// Mitsubishi GX Works2 project: Tetris_20220329   PLC: Q03UDV

PROGRAM 94_TOOLS  // Common Tools
; [Title]P1030 Calculate 16's Field Address
      P1030
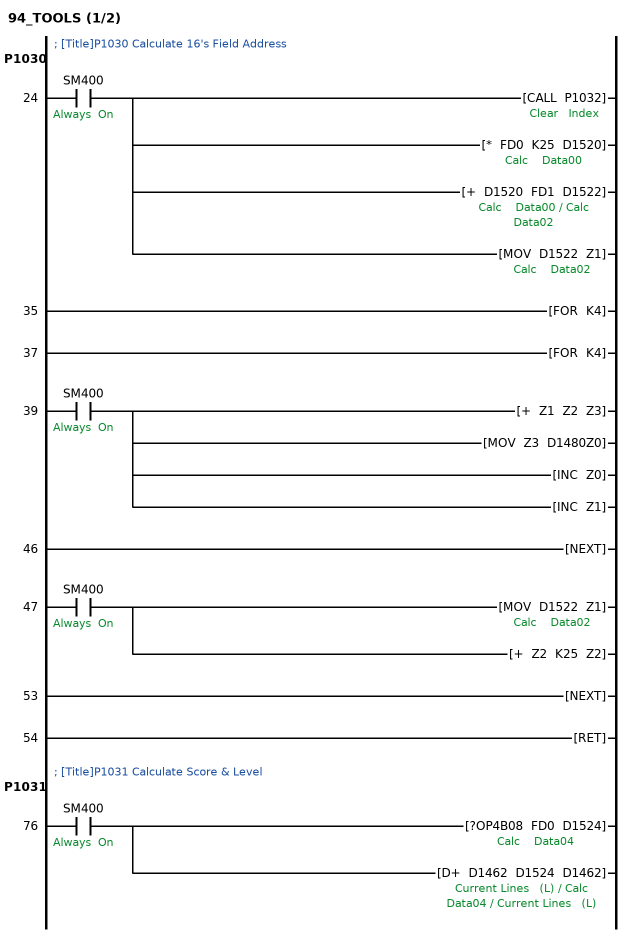
24    LD      SM400  ; Always  On
      CALL    P1032  ; Clear   Index
      *       FD0 K25 D1520  ; Calc    Data00
      +       D1520 FD1 D1522  ; Calc    Data02
      MOV     D1522 Z1
35    FOR     K4
37    FOR     K4
39    LD      SM400  ; Always  On
      +       Z1 Z2 Z3
      MOV     Z3 D1480Z0
      INC     Z0
      INC     Z1
46    NEXT
47    LD      SM400  ; Always  On
      MOV     D1522 Z1
      +       Z2 K25 Z2
53    NEXT
54    RET
; [Title]P1031 Calculate Score & Level
      P1031
76    LD      SM400  ; Always  On
      ?OP4B08 FD0 D1524  ; Calc    Data04
      D+      D1462 D1524 D1462  ; Current Lines   (L)
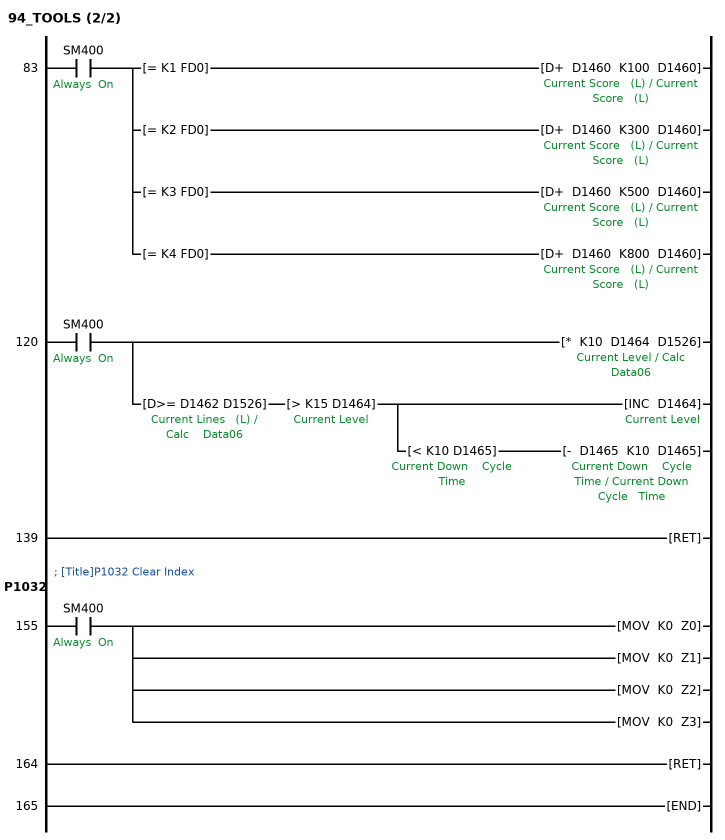
83    LD      SM400  ; Always  On
      MPS
      AND=    K1 FD0
      D+      D1460 K100 D1460  ; Current Score   (L)
      MRD
      AND=    K2 FD0
      D+      D1460 K300 D1460
      MRD
      AND=    K3 FD0
      D+      D1460 K500 D1460
      MPP
      AND=    K4 FD0
      D+      D1460 K800 D1460
120   LD      SM400  ; Always  On
      *       K10 D1464 D1526  ; Current Level / Calc    Data06
      ANDD>=  D1462 D1526  ; Current Lines   (L) / Calc    Data06
      AND>    K15 D1464  ; Current Level
      INC     D1464
      AND<    K10 D1465  ; Current Down    Cycle   Time
      -       D1465 K10 D1465
139   RET
; [Title]P1032 Clear Index
      P1032
155   LD      SM400  ; Always  On
      MOV     K0 Z0
      MOV     K0 Z1
      MOV     K0 Z2
      MOV     K0 Z3
164   RET
165   END
END_PROGRAM

PROGRAM 02_GAME  // Main Game Control
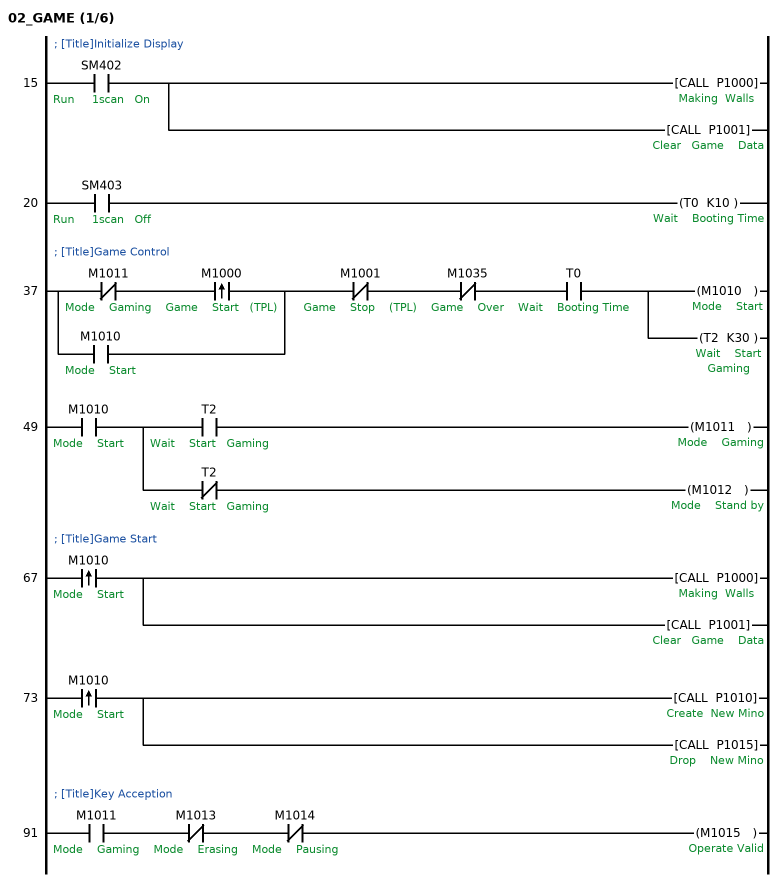
; [Title]Initialize Display
15    LD      SM402  ; Run     1scan   On
      CALL    P1000  ; Making  Walls
      CALL    P1001  ; Clear   Game    Data
20    LD      SM403  ; Run     1scan   Off
      OUT     T0 K10  ; Wait    Booting Time
; [Title]Game Control
37    LDI     M1011  ; Mode    Gaming
      ANDP    M1000  ; Game    Start   (TPL)
      OR      M1010  ; Mode    Start
      ANI     M1001  ; Game    Stop    (TPL)
      ANI     M1035  ; Game    Over
      AND     T0  ; Wait    Booting Time
      OUT     M1010  ; Mode    Start
      OUT     T2 K30  ; Wait    Start   Gaming
49    LD      M1010  ; Mode    Start
      MPS
      AND     T2  ; Wait    Start   Gaming
      OUT     M1011  ; Mode    Gaming
      MPP
      ANI     T2  ; Wait    Start   Gaming
      OUT     M1012  ; Mode    Stand by
; [Title]Game Start
67    LDP     M1010  ; Mode    Start
      CALL    P1000
      CALL    P1001
73    LDP     M1010  ; Mode    Start
      CALL    P1010  ; Create  New Mino
      CALL    P1015  ; Drop    New Mino
; [Title]Key Acception
91    LD      M1011  ; Mode    Gaming
      ANI     M1013  ; Mode    Erasing
      ANI     M1014  ; Mode    Pausing
      OUT     M1015  ; Operate Valid
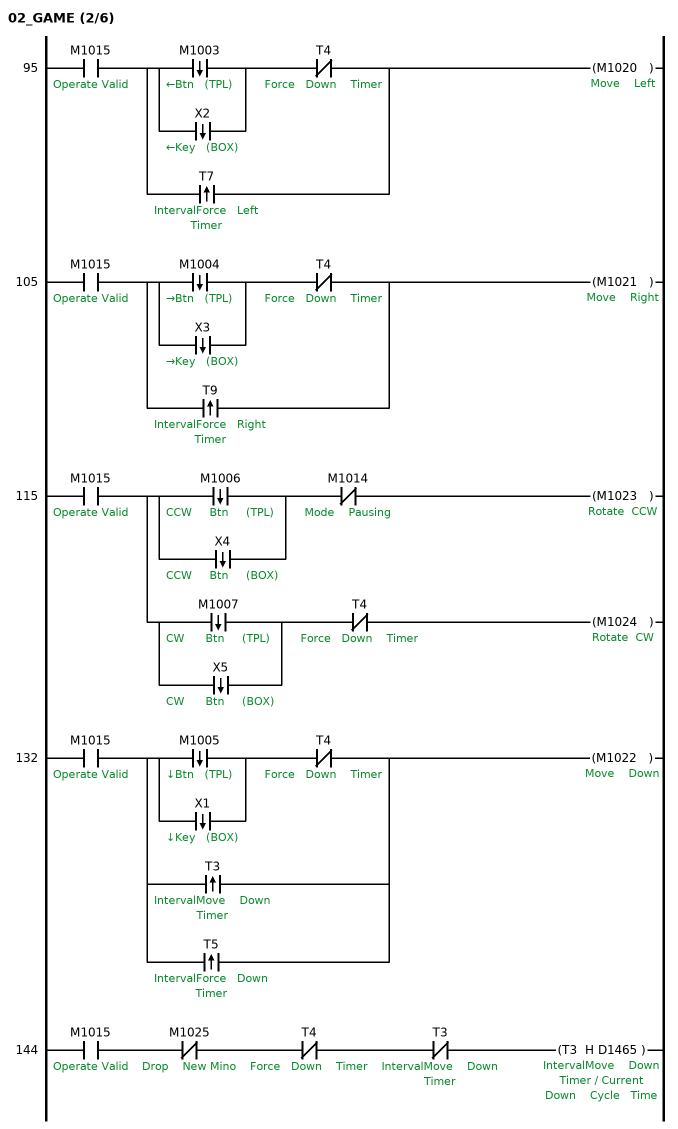
95    LD      M1015  ; Operate Valid
      LDF     M1003  ; ←Btn   (TPL)
      ORF     X2  ; ←Key   (BOX)
      ANI     T4  ; Force   Down    Timer
      ORP     T7  ; IntervalForce   Left    Timer
      ANB
      OUT     M1020  ; Move    Left
105   LD      M1015  ; Operate Valid
      LDF     M1004  ; →Btn   (TPL)
      ORF     X3  ; →Key   (BOX)
      ANI     T4  ; Force   Down    Timer
      ORP     T9  ; IntervalForce   Right   Timer
      ANB
      OUT     M1021  ; Move    Right
115   LD      M1015  ; Operate Valid
      MPS
      LDF     M1006  ; CCW     Btn     (TPL)
      ORF     X4  ; CCW     Btn     (BOX)
      ANB
      ANI     M1014  ; Mode    Pausing
      OUT     M1023  ; Rotate  CCW
      MPP
      LDF     M1007  ; CW      Btn     (TPL)
      ORF     X5  ; CW      Btn     (BOX)
      ANB
      ANI     T4  ; Force   Down    Timer
      OUT     M1024  ; Rotate  CW
132   LD      M1015  ; Operate Valid
      LDF     M1005  ; ↓Btn   (TPL)
      ORF     X1  ; ↓Key   (BOX)
      ANI     T4  ; Force   Down    Timer
      ORP     T3  ; IntervalMove    Down    Timer
      ORP     T5  ; IntervalForce   Down    Timer
      ANB
      OUT     M1022  ; Move    Down
144   LD      M1015  ; Operate Valid
      ANI     M1025  ; Drop    New Mino
      ANI     T4  ; Force   Down    Timer
      ANI     T3  ; IntervalMove    Down    Timer
      OUTH    T3 D1465  ; IntervalMove    Down    Timer / Current Down    Cycle   Time
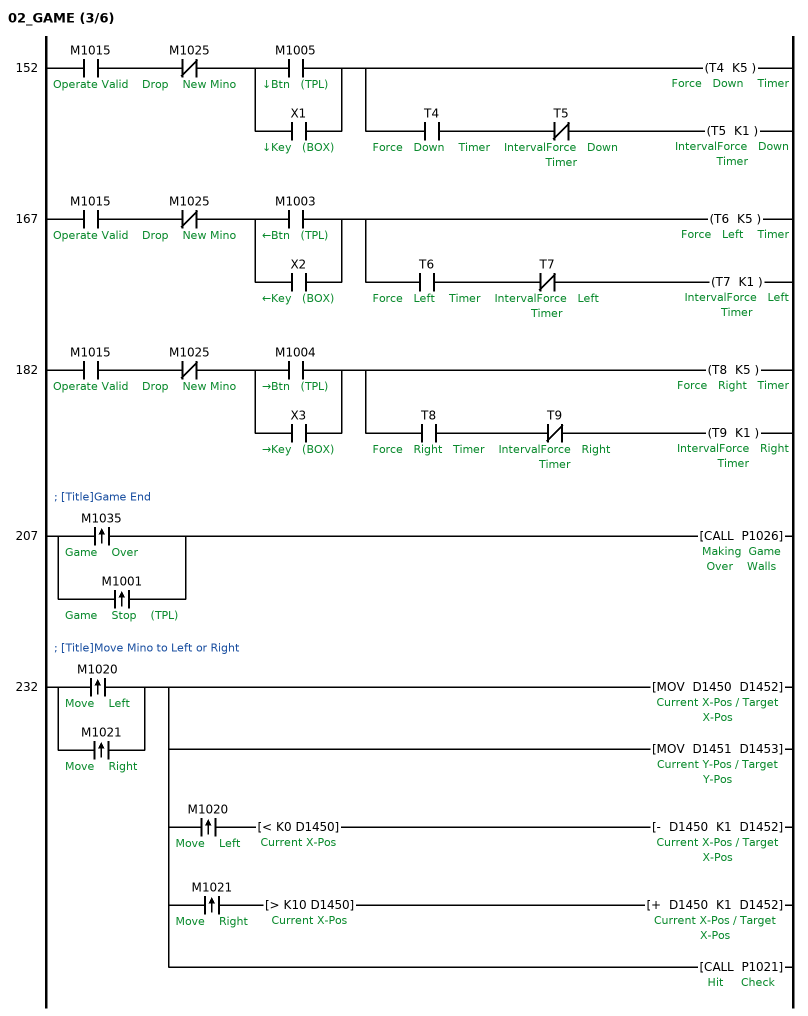
152   LD      M1015  ; Operate Valid
      ANI     M1025  ; Drop    New Mino
      LD      M1005  ; ↓Btn   (TPL)
      OR      X1  ; ↓Key   (BOX)
      ANB
      OUT     T4 K5  ; Force   Down    Timer
      AND     T4  ; Force   Down    Timer
      ANI     T5  ; IntervalForce   Down    Timer
      OUT     T5 K1  ; IntervalForce   Down    Timer
167   LD      M1015  ; Operate Valid
      ANI     M1025  ; Drop    New Mino
      LD      M1003  ; ←Btn   (TPL)
      OR      X2  ; ←Key   (BOX)
      ANB
      OUT     T6 K5  ; Force   Left    Timer
      AND     T6  ; Force   Left    Timer
      ANI     T7  ; IntervalForce   Left    Timer
      OUT     T7 K1  ; IntervalForce   Left    Timer
182   LD      M1015  ; Operate Valid
      ANI     M1025  ; Drop    New Mino
      LD      M1004  ; →Btn   (TPL)
      OR      X3  ; →Key   (BOX)
      ANB
      OUT     T8 K5  ; Force   Right   Timer
      AND     T8  ; Force   Right   Timer
      ANI     T9  ; IntervalForce   Right   Timer
      OUT     T9 K1  ; IntervalForce   Right   Timer
; [Title]Game End
207   LDP     M1035  ; Game    Over
      ORP     M1001  ; Game    Stop    (TPL)
      CALL    P1026  ; Making  Game    Over    Walls
; [Title]Move Mino to Left or Right
232   LDP     M1020  ; Move    Left
      ORP     M1021  ; Move    Right
      MOV     D1450 D1452  ; Current X-Pos / Target  X-Pos
      MOV     D1451 D1453  ; Current Y-Pos / Target  Y-Pos
      MPS
      ANDP    M1020  ; Move    Left
      AND<    K0 D1450  ; Current X-Pos
      -       D1450 K1 D1452
      MRD
      ANDP    M1021  ; Move    Right
      AND>    K10 D1450  ; Current X-Pos
      +       D1450 K1 D1452
      MPP
      CALL    P1021  ; Hit     Check
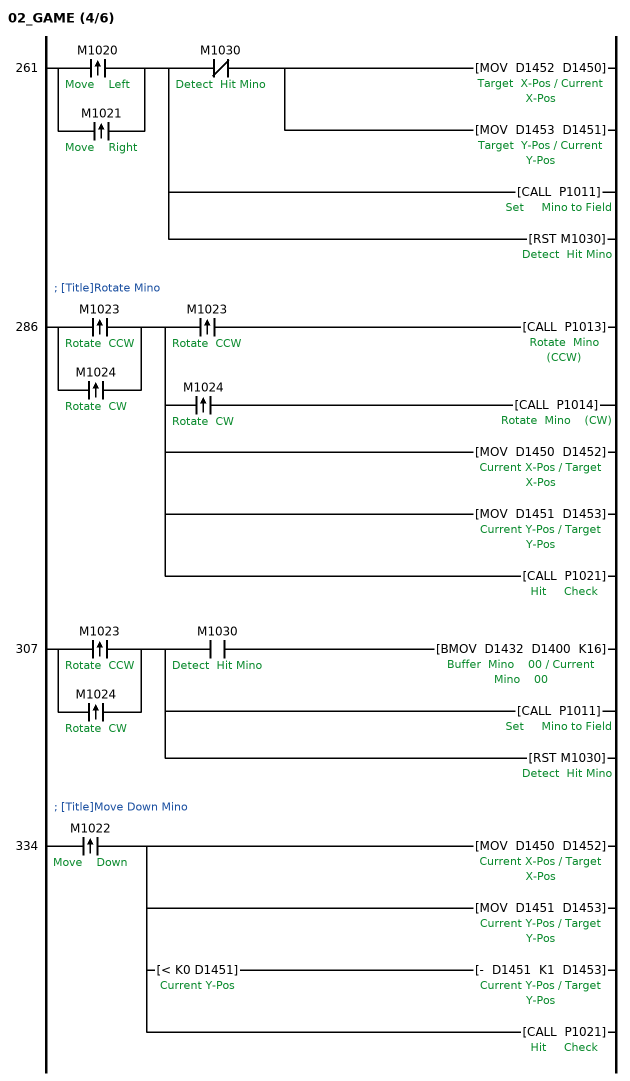
261   LDP     M1020  ; Move    Left
      ORP     M1021  ; Move    Right
      MPS
      ANI     M1030  ; Detect  Hit Mino
      MOV     D1452 D1450
      MOV     D1453 D1451
      MPP
      CALL    P1011  ; Set     Mino to Field
      RST     M1030  ; Detect  Hit Mino
; [Title]Rotate Mino
286   LDP     M1023  ; Rotate  CCW
      ORP     M1024  ; Rotate  CW
      MPS
      ANDP    M1023  ; Rotate  CCW
      CALL    P1013  ; Rotate  Mino    (CCW)
      MRD
      ANDP    M1024  ; Rotate  CW
      CALL    P1014  ; Rotate  Mino    (CW)
      MPP
      MOV     D1450 D1452
      MOV     D1451 D1453
      CALL    P1021
307   LDP     M1023  ; Rotate  CCW
      ORP     M1024  ; Rotate  CW
      MPS
      AND     M1030  ; Detect  Hit Mino
      BMOV    D1432 D1400 K16  ; Buffer  Mino    00 / Current Mino    00
      MPP
      CALL    P1011
      RST     M1030  ; Detect  Hit Mino
; [Title]Move Down Mino
334   LDP     M1022  ; Move    Down
      MOV     D1450 D1452
      MOV     D1451 D1453
      MPS
      AND<    K0 D1451  ; Current Y-Pos
      -       D1451 K1 D1453
      MPP
      CALL    P1021
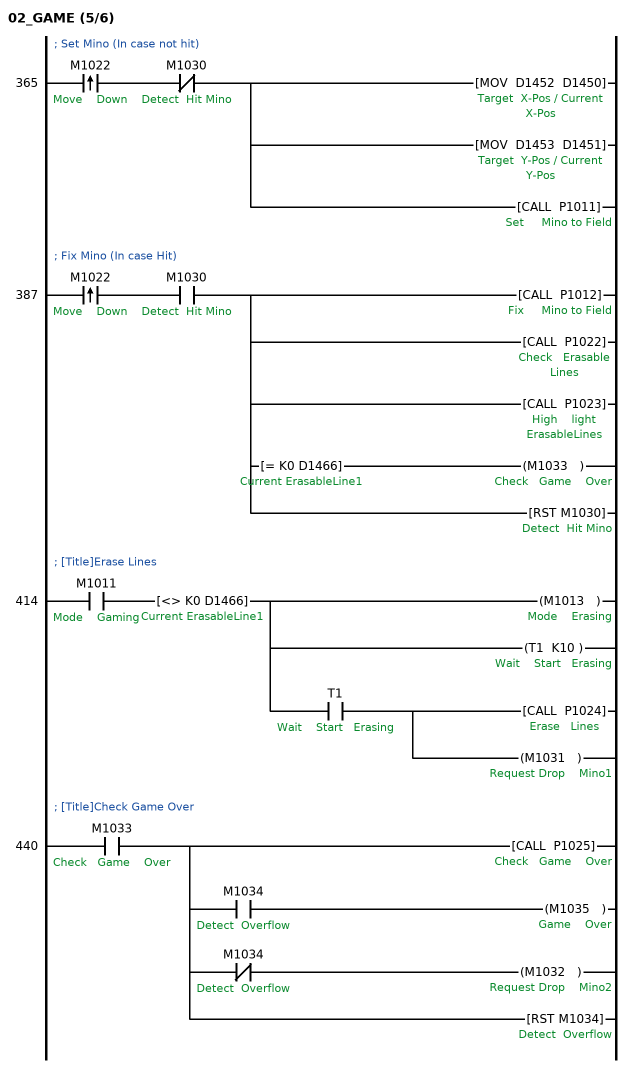
; Set Mino (In case not hit)
365   LDP     M1022  ; Move    Down
      ANI     M1030  ; Detect  Hit Mino
      MOV     D1452 D1450
      MOV     D1453 D1451
      CALL    P1011
; Fix Mino (In case Hit)
387   LDP     M1022  ; Move    Down
      AND     M1030  ; Detect  Hit Mino
      CALL    P1012  ; Fix     Mino to Field
      CALL    P1022  ; Check   ErasableLines
      CALL    P1023  ; High    light   ErasableLines
      MPS
      AND=    K0 D1466  ; Current ErasableLine1
      OUT     M1033  ; Check   Game    Over
      MPP
      RST     M1030  ; Detect  Hit Mino
; [Title]Erase Lines
414   LD      M1011  ; Mode    Gaming
      AND<>   K0 D1466  ; Current ErasableLine1
      OUT     M1013  ; Mode    Erasing
      OUT     T1 K10  ; Wait    Start   Erasing
      AND     T1  ; Wait    Start   Erasing
      CALL    P1024  ; Erase   Lines
      OUT     M1031  ; Request Drop    Mino1
; [Title]Check Game Over
440   LD      M1033  ; Check   Game    Over
      CALL    P1025  ; Check   Game    Over
      MPS
      AND     M1034  ; Detect  Overflow
      OUT     M1035  ; Game    Over
      MRD
      ANI     M1034  ; Detect  Overflow
      OUT     M1032  ; Request Drop    Mino2
      MPP
      RST     M1034  ; Detect  Overflow
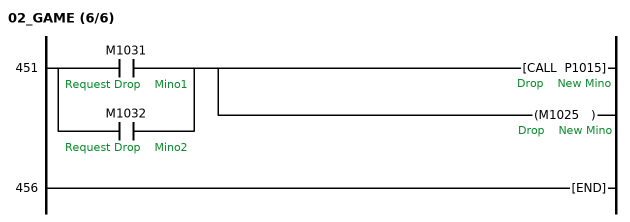
451   LD      M1031  ; Request Drop    Mino1
      OR      M1032  ; Request Drop    Mino2
      CALL    P1015
      OUT     M1025  ; Drop    New Mino
456   END
END_PROGRAM

PROGRAM 91_SETUP  // Setup Condition
; [Title]P1000 Making Walls
; Make Walls and Clear Field
      P1000
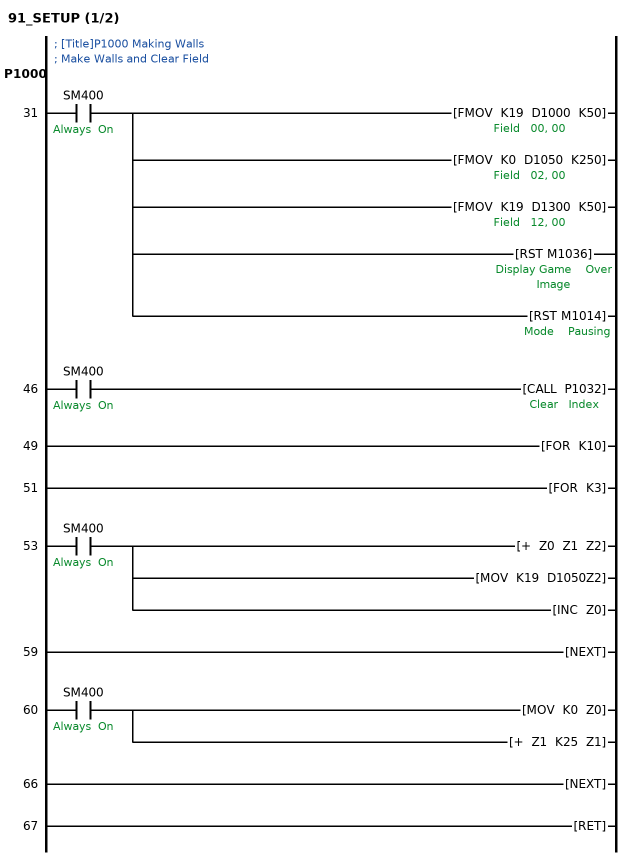
31    LD      SM400  ; Always  On
      FMOV    K19 D1000 K50  ; Field   00, 00
      FMOV    K0 D1050 K250  ; Field   02, 00
      FMOV    K19 D1300 K50  ; Field   12, 00
      RST     M1036  ; Display Game    Over    Image
      RST     M1014  ; Mode    Pausing
46    LD      SM400  ; Always  On
      CALL    P1032  ; Clear   Index
49    FOR     K10
51    FOR     K3
53    LD      SM400  ; Always  On
      +       Z0 Z1 Z2
      MOV     K19 D1050Z2
      INC     Z0
59    NEXT
60    LD      SM400  ; Always  On
      MOV     K0 Z0
      +       Z1 K25 Z1
66    NEXT
67    RET
; [Title]P1001 Clear All Game Data
      P1001
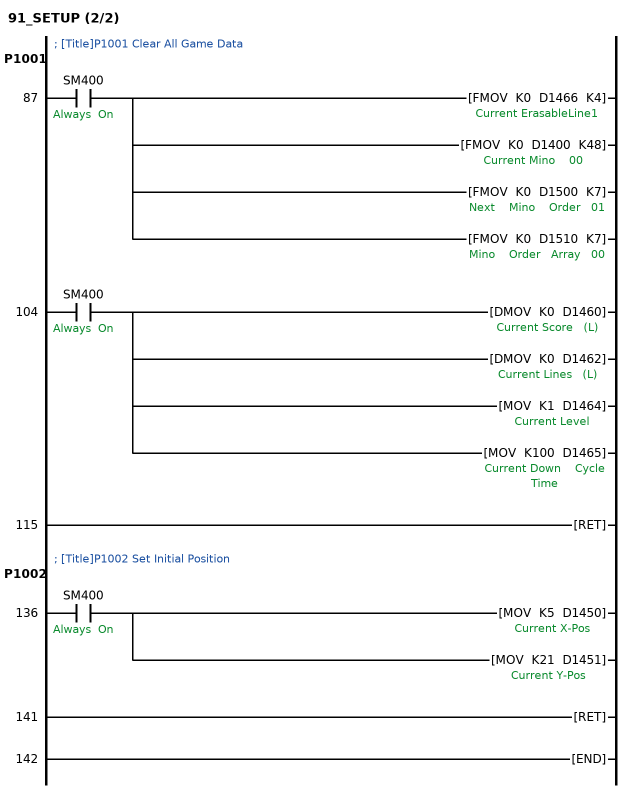
87    LD      SM400  ; Always  On
      FMOV    K0 D1466 K4  ; Current ErasableLine1
      FMOV    K0 D1400 K48  ; Current Mino    00
      FMOV    K0 D1500 K7  ; Next    Mino    Order   01
      FMOV    K0 D1510 K7  ; Mino    Order   Array   00
104   LD      SM400  ; Always  On
      DMOV    K0 D1460  ; Current Score   (L)
      DMOV    K0 D1462  ; Current Lines   (L)
      MOV     K1 D1464  ; Current Level
      MOV     K100 D1465  ; Current Down    Cycle   Time
115   RET
; [Title]P1002 Set Initial Position
      P1002
136   LD      SM400  ; Always  On
      MOV     K5 D1450  ; Current X-Pos
      MOV     K21 D1451  ; Current Y-Pos
141   RET
142   END
END_PROGRAM

PROGRAM 92_MINO  // Manage Mino
; [Title]P1010 Create New Mino
; Make New Mino Order & Copy Mino Data to Reserve Mino Area
      P1010
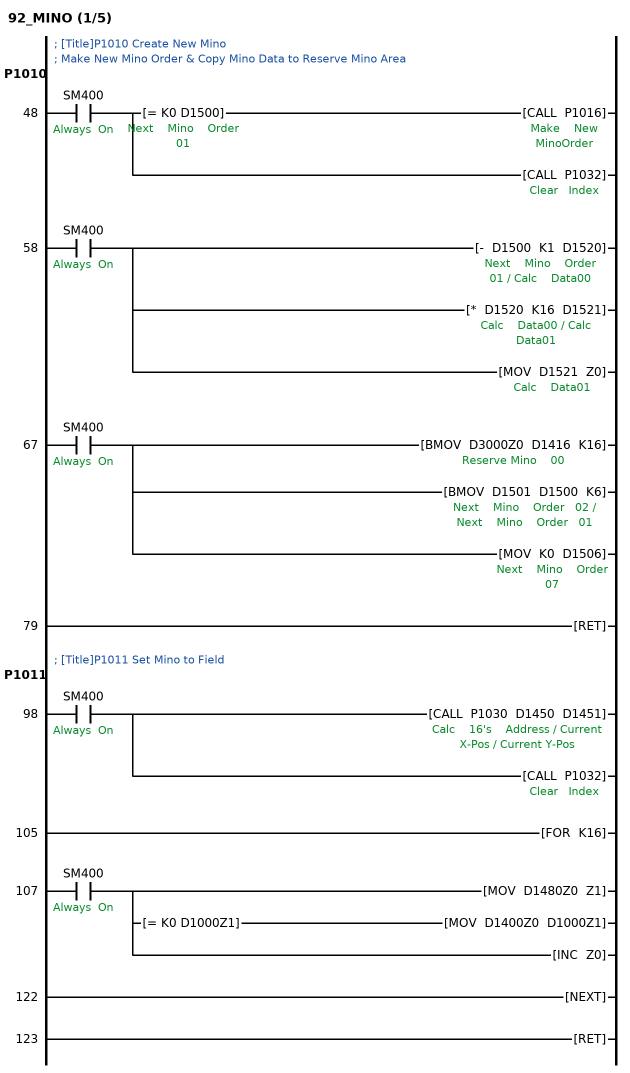
48    LD      SM400  ; Always  On
      MPS
      AND=    K0 D1500  ; Next    Mino    Order   01
      CALL    P1016  ; Make    New MinoOrder
      MPP
      CALL    P1032  ; Clear   Index
58    LD      SM400  ; Always  On
      -       D1500 K1 D1520  ; Calc    Data00
      *       D1520 K16 D1521  ; Calc    Data01
      MOV     D1521 Z0
67    LD      SM400  ; Always  On
      BMOV    D3000Z0 D1416 K16  ; Reserve Mino    00
      BMOV    D1501 D1500 K6  ; Next    Mino    Order   02
      MOV     K0 D1506  ; Next    Mino    Order   07
79    RET
; [Title]P1011 Set Mino to Field
      P1011
98    LD      SM400  ; Always  On
      CALL    P1030 D1450 D1451  ; Calc    16's    Address / Current X-Pos / Current Y-Pos
      CALL    P1032
105   FOR     K16
107   LD      SM400  ; Always  On
      MOV     D1480Z0 Z1
      MPS
      AND=    K0 D1000Z1
      MOV     D1400Z0 D1000Z1
      MPP
      INC     Z0
122   NEXT
123   RET
; [Title]P1012 Fix Mino to Field
      P1012
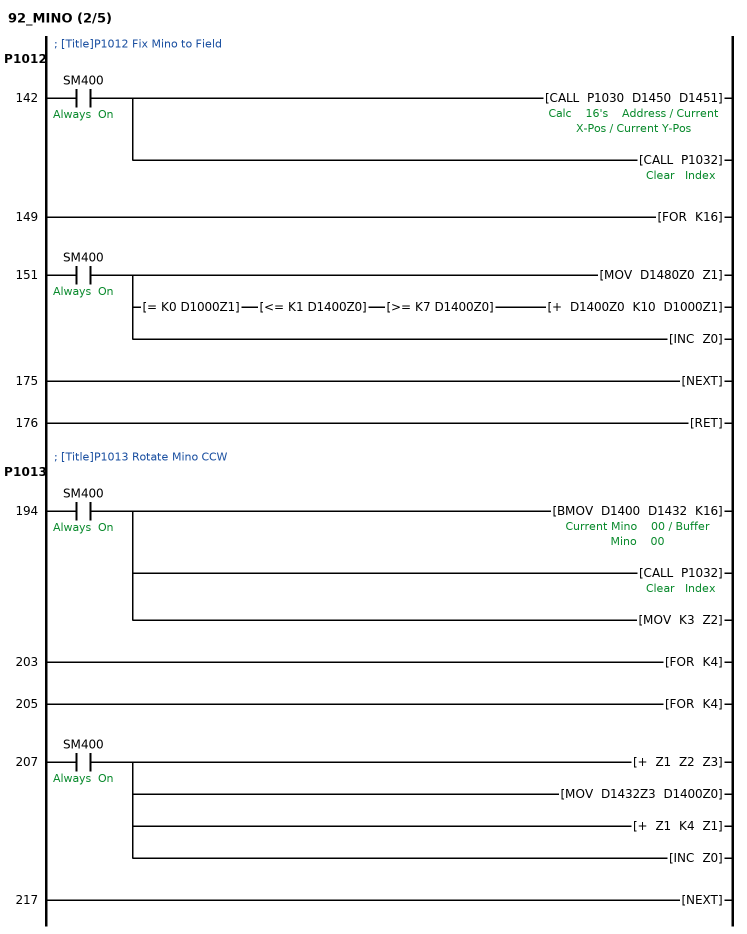
142   LD      SM400  ; Always  On
      CALL    P1030 D1450 D1451
      CALL    P1032
149   FOR     K16
151   LD      SM400  ; Always  On
      MOV     D1480Z0 Z1
      MPS
      AND=    K0 D1000Z1
      AND<=   K1 D1400Z0
      AND>=   K7 D1400Z0
      +       D1400Z0 K10 D1000Z1
      MPP
      INC     Z0
175   NEXT
176   RET
; [Title]P1013 Rotate Mino CCW
      P1013
194   LD      SM400  ; Always  On
      BMOV    D1400 D1432 K16  ; Current Mino    00 / Buffer  Mino    00
      CALL    P1032
      MOV     K3 Z2
203   FOR     K4
205   FOR     K4
207   LD      SM400  ; Always  On
      +       Z1 Z2 Z3
      MOV     D1432Z3 D1400Z0
      +       Z1 K4 Z1
      INC     Z0
217   NEXT
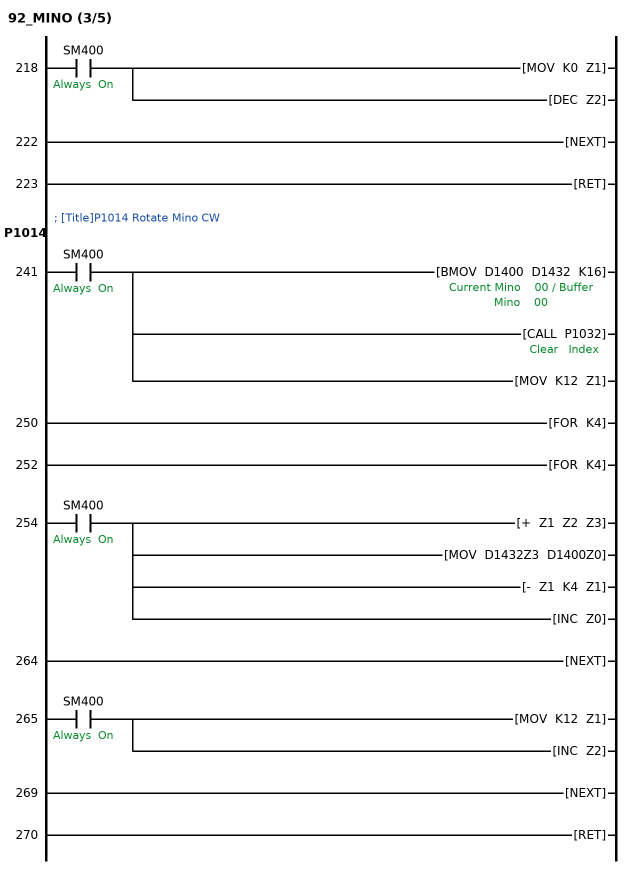
218   LD      SM400  ; Always  On
      MOV     K0 Z1
      DEC     Z2
222   NEXT
223   RET
; [Title]P1014 Rotate Mino CW
      P1014
241   LD      SM400  ; Always  On
      BMOV    D1400 D1432 K16
      CALL    P1032
      MOV     K12 Z1
250   FOR     K4
252   FOR     K4
254   LD      SM400  ; Always  On
      +       Z1 Z2 Z3
      MOV     D1432Z3 D1400Z0
      -       Z1 K4 Z1
      INC     Z0
264   NEXT
265   LD      SM400  ; Always  On
      MOV     K12 Z1
      INC     Z2
269   NEXT
270   RET
; [Title]P1015 Drop New Mino to Field
      P1015
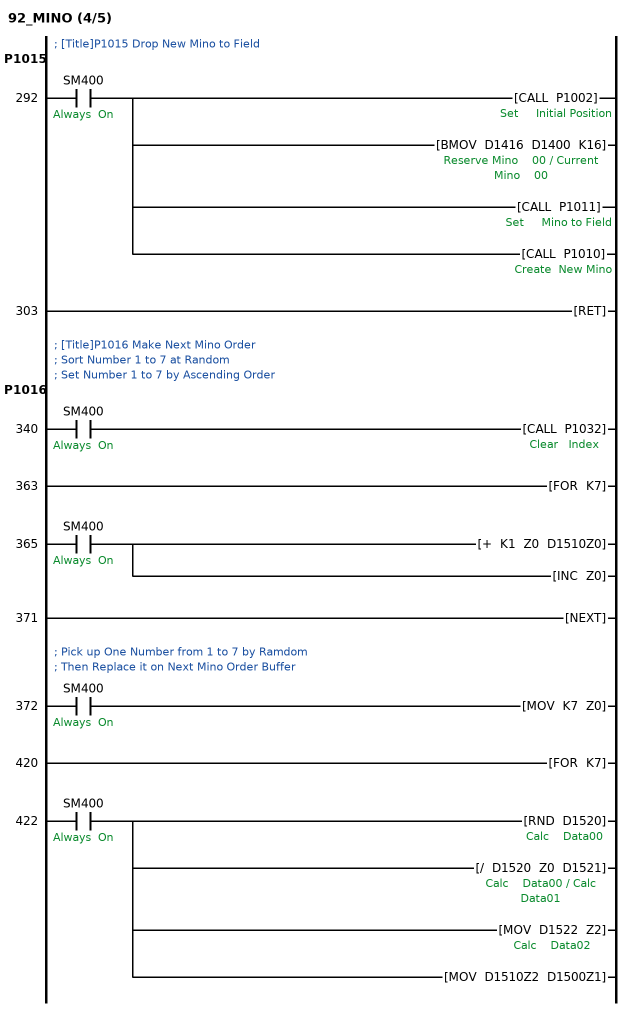
292   LD      SM400  ; Always  On
      CALL    P1002  ; Set     Initial Position
      BMOV    D1416 D1400 K16
      CALL    P1011  ; Set     Mino to Field
      CALL    P1010  ; Create  New Mino
303   RET
; [Title]P1016 Make Next Mino Order
; Sort Number 1 to 7 at Random
      P1016
340   LD      SM400  ; Always  On
      CALL    P1032
; Set Number 1 to 7 by Ascending Order
363   FOR     K7
365   LD      SM400  ; Always  On
      +       K1 Z0 D1510Z0
      INC     Z0
371   NEXT
372   LD      SM400  ; Always  On
      MOV     K7 Z0
; Pick up One Number from 1 to 7 by Ramdom
; Then Replace it on Next Mino Order Buffer
420   FOR     K7
422   LD      SM400  ; Always  On
      RND     D1520
      /       D1520 Z0 D1521
      MOV     D1522 Z2  ; Calc    Data02
      MOV     D1510Z2 D1500Z1
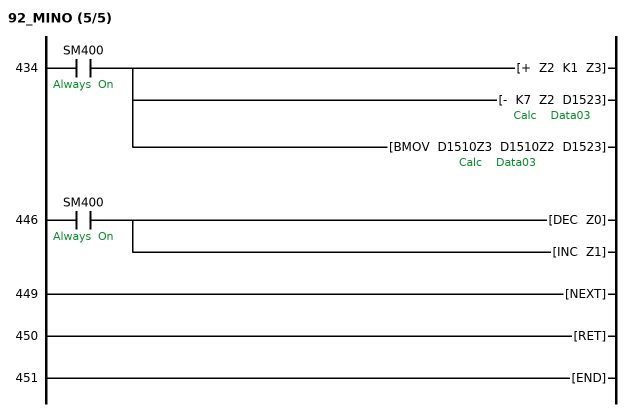
434   LD      SM400  ; Always  On
      +       Z2 K1 Z3
      -       K7 Z2 D1523  ; Calc    Data03
      BMOV    D1510Z3 D1510Z2 D1523
446   LD      SM400  ; Always  On
      DEC     Z0
      INC     Z1
449   NEXT
450   RET
451   END
END_PROGRAM

PROGRAM 93_FIELD  // Manage Field
; [Title]P1020 Clear Field Blocks
; Only Clear Floating Blocks (Not Fixed Blocks)
      P1020
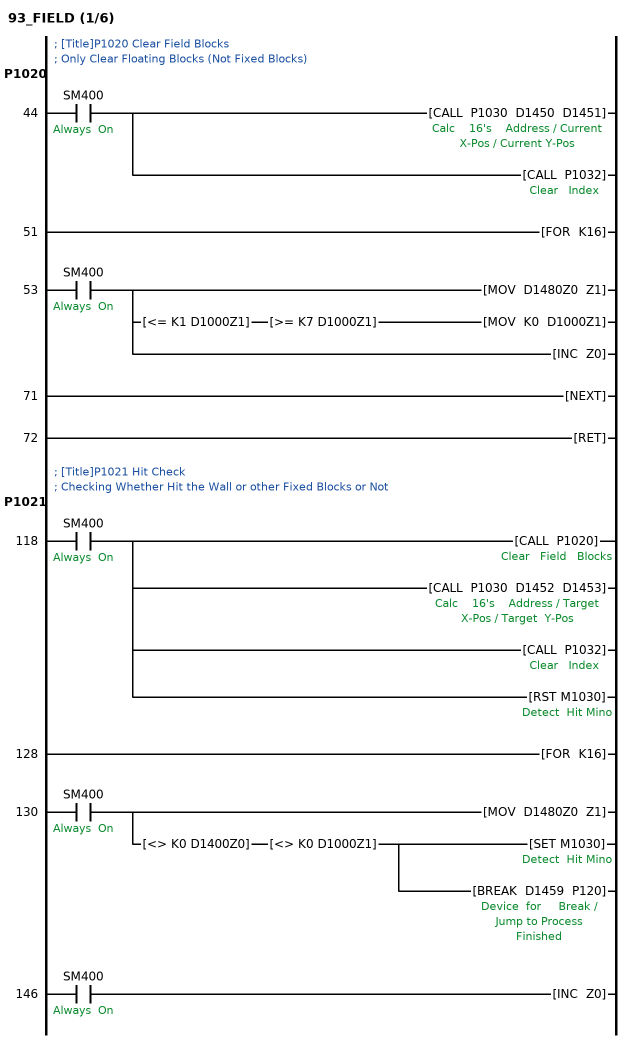
44    LD      SM400  ; Always  On
      CALL    P1030 D1450 D1451  ; Calc    16's    Address / Current X-Pos / Current Y-Pos
      CALL    P1032  ; Clear   Index
51    FOR     K16
53    LD      SM400  ; Always  On
      MOV     D1480Z0 Z1
      MPS
      AND<=   K1 D1000Z1
      AND>=   K7 D1000Z1
      MOV     K0 D1000Z1
      MPP
      INC     Z0
71    NEXT
72    RET
; [Title]P1021 Hit Check
; Checking Whether Hit the Wall or other Fixed Blocks or Not
      P1021
118   LD      SM400  ; Always  On
      CALL    P1020  ; Clear   Field   Blocks
      CALL    P1030 D1452 D1453  ; Target  X-Pos / Target  Y-Pos
      CALL    P1032
      RST     M1030  ; Detect  Hit Mino
128   FOR     K16
130   LD      SM400  ; Always  On
      MOV     D1480Z0 Z1
      AND<>   K0 D1400Z0
      AND<>   K0 D1000Z1
      SET     M1030  ; Detect  Hit Mino
      BREAK   D1459 P120  ; Device  for     Break / Jump to Process Finished
146   LD      SM400  ; Always  On
      INC     Z0
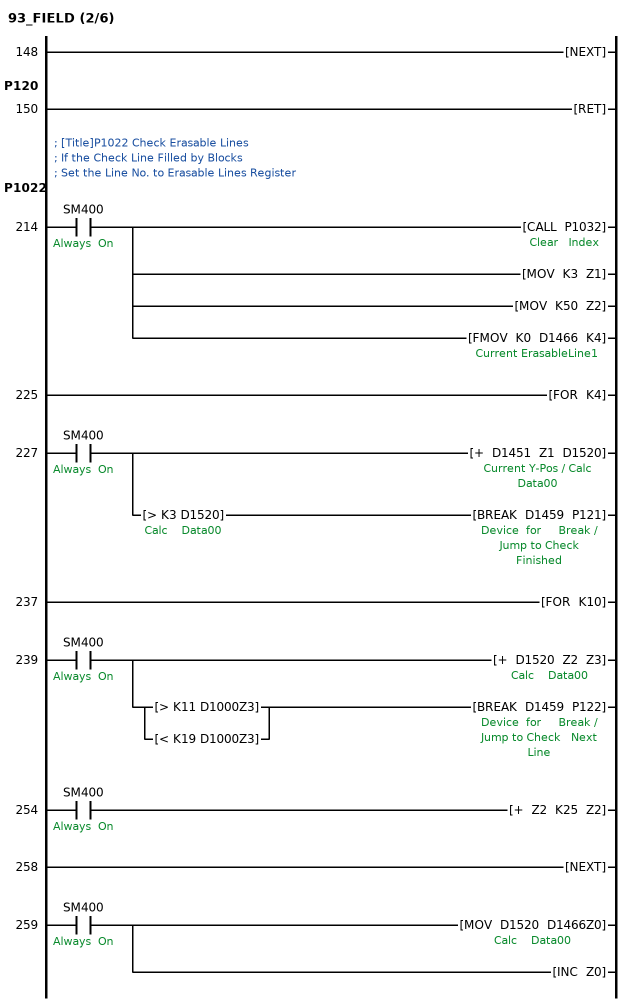
148   NEXT
      P120
150   RET
; [Title]P1022 Check Erasable Lines
; If the Check Line Filled by Blocks
; Set the Line No. to Erasable Lines Register
      P1022
214   LD      SM400  ; Always  On
      CALL    P1032
      MOV     K3 Z1
      MOV     K50 Z2
      FMOV    K0 D1466 K4  ; Current ErasableLine1
225   FOR     K4
227   LD      SM400  ; Always  On
      +       D1451 Z1 D1520  ; Calc    Data00
      AND>    K3 D1520  ; Calc    Data00
      BREAK   D1459 P121  ; Jump to Check   Finished
237   FOR     K10
239   LD      SM400  ; Always  On
      +       D1520 Z2 Z3
      LD>     K11 D1000Z3
      OR<     K19 D1000Z3
      ANB
      BREAK   D1459 P122  ; Jump to Check   Next    Line
254   LD      SM400  ; Always  On
      +       Z2 K25 Z2
258   NEXT
259   LD      SM400  ; Always  On
      MOV     D1520 D1466Z0
      INC     Z0
      P122
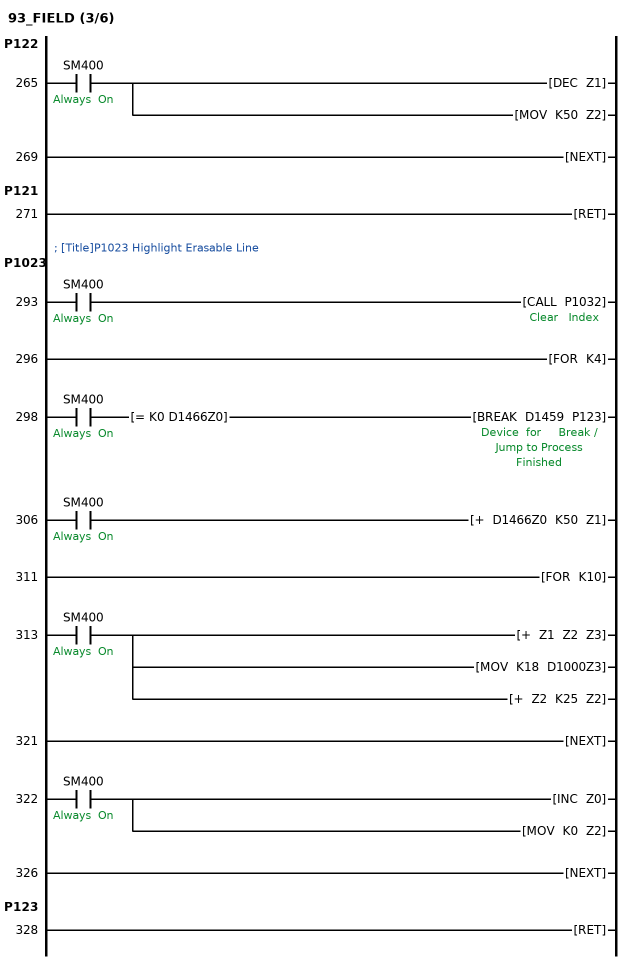
265   LD      SM400  ; Always  On
      DEC     Z1
      MOV     K50 Z2
269   NEXT
      P121
271   RET
; [Title]P1023 Highlight Erasable Line
      P1023
293   LD      SM400  ; Always  On
      CALL    P1032
296   FOR     K4
298   LD      SM400  ; Always  On
      AND=    K0 D1466Z0
      BREAK   D1459 P123  ; Jump to Process Finished
306   LD      SM400  ; Always  On
      +       D1466Z0 K50 Z1
311   FOR     K10
313   LD      SM400  ; Always  On
      +       Z1 Z2 Z3
      MOV     K18 D1000Z3
      +       Z2 K25 Z2
321   NEXT
322   LD      SM400  ; Always  On
      INC     Z0
      MOV     K0 Z2
326   NEXT
      P123
328   RET
; [Title]P1024 Erase Lines
      P1024
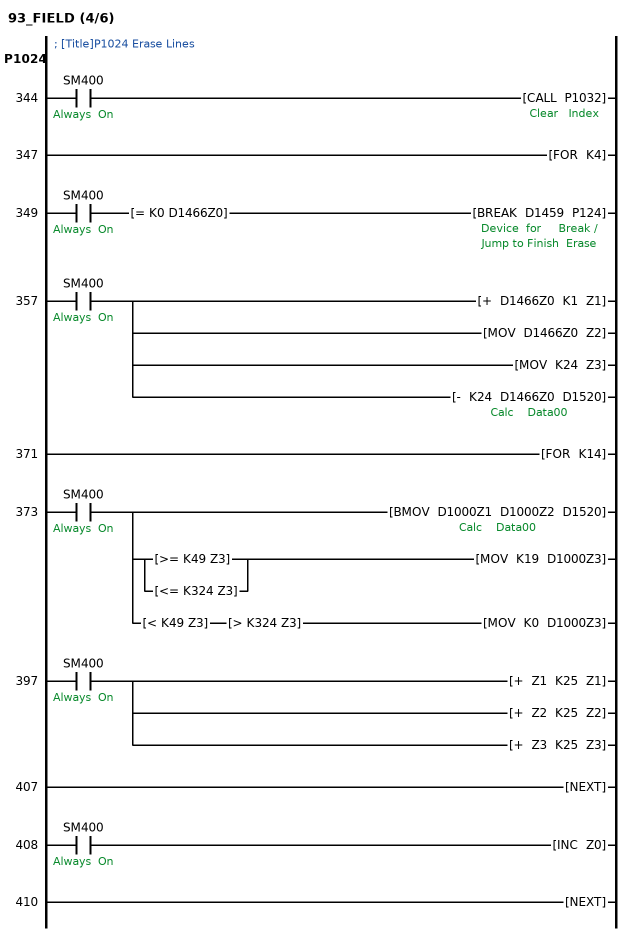
344   LD      SM400  ; Always  On
      CALL    P1032
347   FOR     K4
349   LD      SM400  ; Always  On
      AND=    K0 D1466Z0
      BREAK   D1459 P124  ; Jump to Finish  Erase
357   LD      SM400  ; Always  On
      +       D1466Z0 K1 Z1
      MOV     D1466Z0 Z2
      MOV     K24 Z3
      -       K24 D1466Z0 D1520
371   FOR     K14
373   LD      SM400  ; Always  On
      BMOV    D1000Z1 D1000Z2 D1520
      MPS
      LD>=    K49 Z3
      OR<=    K324 Z3
      ANB
      MOV     K19 D1000Z3
      MPP
      AND<    K49 Z3
      AND>    K324 Z3
      MOV     K0 D1000Z3
397   LD      SM400  ; Always  On
      +       Z1 K25 Z1
      +       Z2 K25 Z2
      +       Z3 K25 Z3
407   NEXT
408   LD      SM400  ; Always  On
      INC     Z0
410   NEXT
      P124
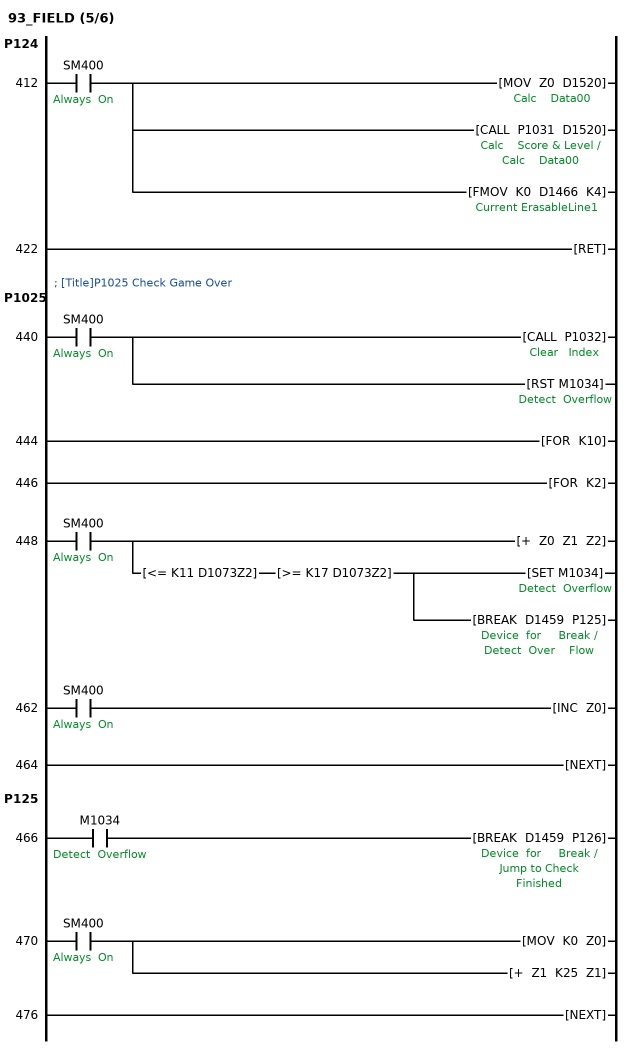
412   LD      SM400  ; Always  On
      MOV     Z0 D1520
      CALL    P1031 D1520  ; Calc    Score & Level
      FMOV    K0 D1466 K4
422   RET
; [Title]P1025 Check Game Over
      P1025
440   LD      SM400  ; Always  On
      CALL    P1032
      RST     M1034  ; Detect  Overflow
444   FOR     K10
446   FOR     K2
448   LD      SM400  ; Always  On
      +       Z0 Z1 Z2
      AND<=   K11 D1073Z2
      AND>=   K17 D1073Z2
      SET     M1034  ; Detect  Overflow
      BREAK   D1459 P125  ; Detect  Over    Flow
462   LD      SM400  ; Always  On
      INC     Z0
464   NEXT
      P125
466   LD      M1034  ; Detect  Overflow
      BREAK   D1459 P126  ; Jump to Check   Finished
470   LD      SM400  ; Always  On
      MOV     K0 Z0
      +       Z1 K25 Z1
476   NEXT
      P126
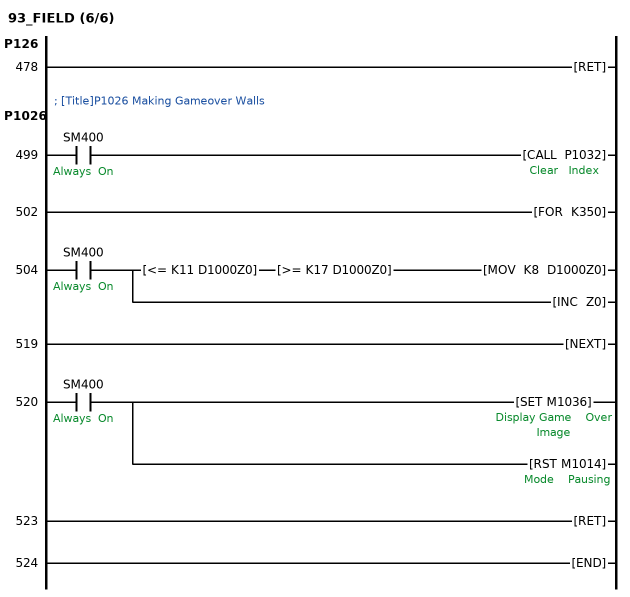
478   RET
; [Title]P1026 Making Gameover Walls
      P1026
499   LD      SM400  ; Always  On
      CALL    P1032
502   FOR     K350
504   LD      SM400  ; Always  On
      MPS
      AND<=   K11 D1000Z0
      AND>=   K17 D1000Z0
      MOV     K8 D1000Z0
      MPP
      INC     Z0
519   NEXT
520   LD      SM400  ; Always  On
      SET     M1036  ; Display Game    Over    Image
      RST     M1014  ; Mode    Pausing
523   RET
524   END
END_PROGRAM

PROGRAM 01_INIT  // Initializing Data
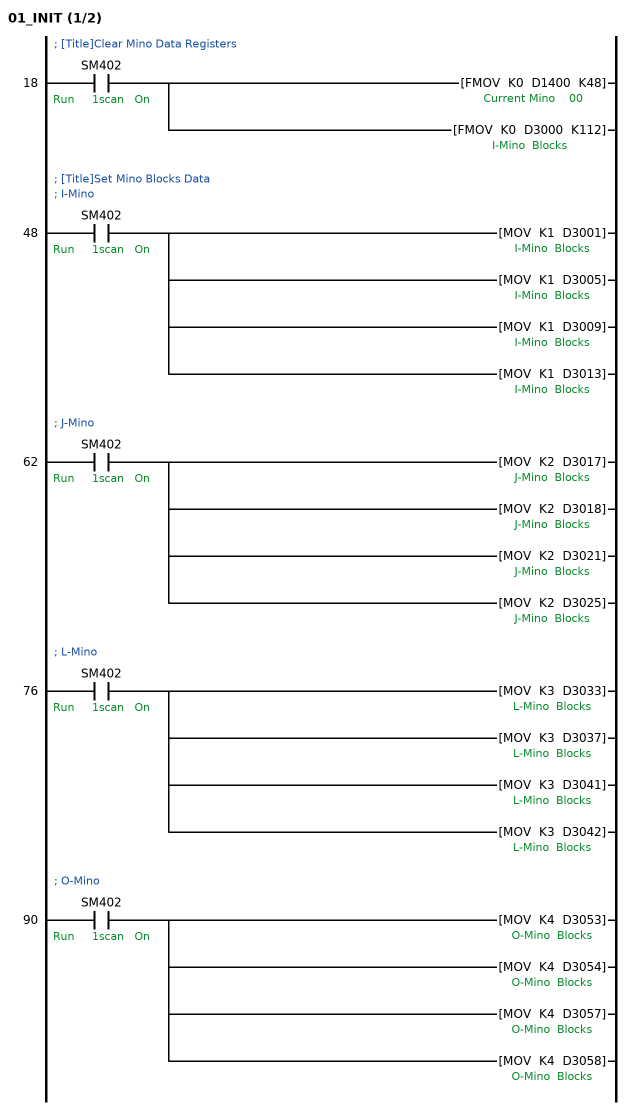
; [Title]Clear Mino Data Registers
18    LD      SM402  ; Run     1scan   On
      FMOV    K0 D1400 K48  ; Current Mino    00
      FMOV    K0 D3000 K112  ; I-Mino  Blocks
; [Title]Set Mino Blocks Data
; I-Mino
48    LD      SM402  ; Run     1scan   On
      MOV     K1 D3001  ; I-Mino  Blocks
      MOV     K1 D3005  ; I-Mino  Blocks
      MOV     K1 D3009  ; I-Mino  Blocks
      MOV     K1 D3013  ; I-Mino  Blocks
; J-Mino
62    LD      SM402  ; Run     1scan   On
      MOV     K2 D3017  ; J-Mino  Blocks
      MOV     K2 D3018  ; J-Mino  Blocks
      MOV     K2 D3021  ; J-Mino  Blocks
      MOV     K2 D3025  ; J-Mino  Blocks
; L-Mino
76    LD      SM402  ; Run     1scan   On
      MOV     K3 D3033  ; L-Mino  Blocks
      MOV     K3 D3037  ; L-Mino  Blocks
      MOV     K3 D3041  ; L-Mino  Blocks
      MOV     K3 D3042  ; L-Mino  Blocks
; O-Mino
90    LD      SM402  ; Run     1scan   On
      MOV     K4 D3053  ; O-Mino  Blocks
      MOV     K4 D3054  ; O-Mino  Blocks
      MOV     K4 D3057  ; O-Mino  Blocks
      MOV     K4 D3058  ; O-Mino  Blocks
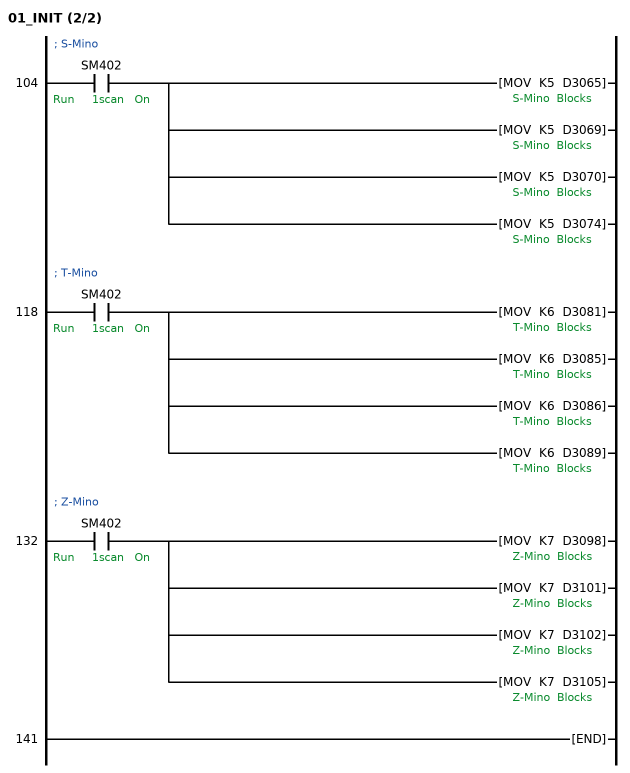
; S-Mino
104   LD      SM402  ; Run     1scan   On
      MOV     K5 D3065  ; S-Mino  Blocks
      MOV     K5 D3069  ; S-Mino  Blocks
      MOV     K5 D3070  ; S-Mino  Blocks
      MOV     K5 D3074  ; S-Mino  Blocks
; T-Mino
118   LD      SM402  ; Run     1scan   On
      MOV     K6 D3081  ; T-Mino  Blocks
      MOV     K6 D3085  ; T-Mino  Blocks
      MOV     K6 D3086  ; T-Mino  Blocks
      MOV     K6 D3089  ; T-Mino  Blocks
; Z-Mino
132   LD      SM402  ; Run     1scan   On
      MOV     K7 D3098  ; Z-Mino  Blocks
      MOV     K7 D3101  ; Z-Mino  Blocks
      MOV     K7 D3102  ; Z-Mino  Blocks
      MOV     K7 D3105  ; Z-Mino  Blocks
141   END
END_PROGRAM

PROGRAM 11_DEBUG  // Test Function for Debug
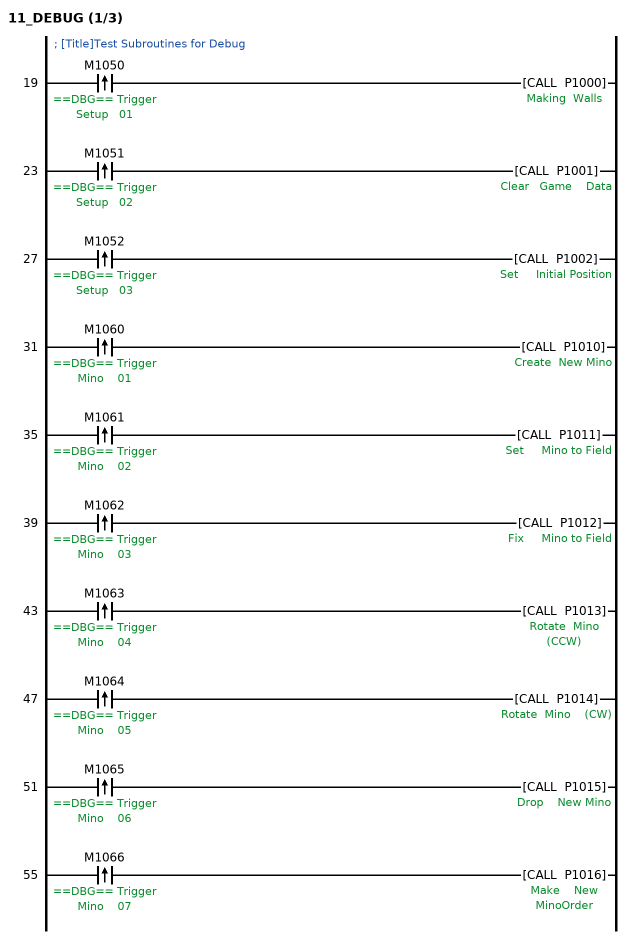
; [Title]Test Subroutines for Debug
19    LDP     M1050  ; ==DBG== Trigger Setup   01
      CALL    P1000  ; Making  Walls
23    LDP     M1051  ; ==DBG== Trigger Setup   02
      CALL    P1001  ; Clear   Game    Data
27    LDP     M1052  ; ==DBG== Trigger Setup   03
      CALL    P1002  ; Set     Initial Position
31    LDP     M1060  ; ==DBG== Trigger Mino    01
      CALL    P1010  ; Create  New Mino
35    LDP     M1061  ; ==DBG== Trigger Mino    02
      CALL    P1011  ; Set     Mino to Field
39    LDP     M1062  ; ==DBG== Trigger Mino    03
      CALL    P1012  ; Fix     Mino to Field
43    LDP     M1063  ; ==DBG== Trigger Mino    04
      CALL    P1013  ; Rotate  Mino    (CCW)
47    LDP     M1064  ; ==DBG== Trigger Mino    05
      CALL    P1014  ; Rotate  Mino    (CW)
51    LDP     M1065  ; ==DBG== Trigger Mino    06
      CALL    P1015  ; Drop    New Mino
55    LDP     M1066  ; ==DBG== Trigger Mino    07
      CALL    P1016  ; Make    New MinoOrder
